// TIA Portal V19 export
FUNCTION "PROG_SELECT_FILLER" : Void   // FC91, STL
TITLE = Program selecter for CIP filler
{ S7_Optimized_Access := 'TRUE' }
NAME : CIP_PROG
// stored: AutoNumber false
BEGIN

NETWORK
TITLE = 
// Update CIP status on OP25 display
      AN    "S0 FILLER";
      R     "Tag_94";
      R     "Tag_95";
      R     "Tag_96";
      R     "Tag_97";
      R     "Tag_98";
      JC    C001;

//    Final rinse
      A     "S40 FILLER";
      O     "S41 FILLER";
      O     "S42 FILLER";
      O     "S43 FILLER";
      O     "S44 FILLER";
      O     "S45 FILLER";
      O     "S46 FILLER";
      O     "S47 FILLER";
      O     "S48 FILLER";
      O     "S49 FILLER";
      R     "Tag_94";
      R     "Tag_95";
      R     "Tag_96";
      R     "Tag_97";
      S     "Tag_98";
      JC    C001;

//    Acid
      A     "S30 FILLER";
      O     "S31 FILLER";
      O     "S32 FILLER";
      O     "S33 FILLER";
      O     "S34 FILLER";
      O     "S35 FILLER";
      O     "S36 FILLER";
      O     "S37 FILLER";
      O     "S38 FILLER";
      O     "S39 FILLER";
      R     "Tag_94";
      R     "Tag_95";
      R     "Tag_96";
      S     "Tag_97";
      R     "Tag_98";
      JC    C001;

//    Middel rinse
      A     "S20 FILLER";
      O     "S21 FILLER";
      O     "S22 FILLER";
      O     "S23 FILLER";
      O     "S24 FILLER";
      O     "S25 FILLER";
      O     "S26 FILLER";
      O     "S27 FILLER";
      O     "S28 FILLER";
      O     "S29 FILLER";
      R     "Tag_94";
      R     "Tag_95";
      S     "Tag_96";
      R     "Tag_97";
      R     "Tag_98";
      JC    C001;

//    Caustic
      A     "S10 FILLER";
      O     "S11 FILLER";
      O     "S12 FILLER";
      O     "S13 FILLER";
      O     "S14 FILLER";
      O     "S15 FILLER";
      O     "S16 FILLER";
      O     "S17 FILLER";
      O     "S18 FILLER";
      O     "S19 FILLER";
      R     "Tag_94";
      S     "Tag_95";
      R     "Tag_96";
      R     "Tag_97";
      R     "Tag_98";
      JC    C001;

//    Pre Rinse
      A     "S0 FILLER";
      O     "S1 FILLER";
      O     "S2 FILLER";
      O     "S3 FILLER";
      O     "S4 FILLER";
      O     "S5 FILLER";
      O     "S6 FILLER";
      O     "S7 FILLER";
      O     "S8 FILLER";
      O     "S9 FILLER";
      S     "Tag_94";
      R     "Tag_95";
      R     "Tag_96";
      R     "Tag_97";
      R     "Tag_98";
      JC    C001;

C001: NOP   0;


NETWORK
TITLE = PROGRAM SELECT 1 CIP FILLER
// Check program select for CIP filler
      A     "S0 FILLER";
      BEC;

      A     "PROG_1_SELECTED";
      S     "CIP_PROG_1";
      R     "CIP_PROG_2";
      R     "CIP_PROG_3";
      L     1;
      T     "Setpoints".ProgCIPFiller;  // "DB SETPOINTS".ProgCIPFiller
      BEC;

      A     "PROG_2_SELECTED";
      S     "CIP_PROG_2";
      R     "CIP_PROG_1";
      R     "CIP_PROG_3";
      L     2;
      T     "Setpoints".ProgCIPFiller;  //"DB SETPOINTS".ProgCIPFiller
      BEC;

      A     "PROG_3_SELECTED";
      S     "CIP_PROG_3";
      R     "CIP_PROG_1";
      R     "CIP_PROG_2";
      L     3;
      T     "Setpoints".ProgCIPFiller;  // "DB SETPOINTS".ProgCIPFiller
      BEC;

      AN    "S0 FILLER";
      R     "CIP_PROG_1";
      R     "CIP_PROG_2";
      S     "CIP_PROG_3";
      L     0;
      T     "Setpoints".ProgCIPFiller;  // "DB SETPOINTS".ProgCIPFiller
      BEU;

END_FUNCTION
